//enum of states
{attribute 'strict'}
{attribute 'to_string'}
{attribute 'qualified_only'}
TYPE eTMP :
(
	TotalReset,
	InitCyl,
	InitSrv,
	InitCamQuickFocus,
	InitCamLoadJob,
	Rest,
	SrvPosStart,
	SrvPosStartInterl,
	SrvPosEnd,
	SrvPosEndIntrl,
	CylOut,
	CylIn,
	MtrStartFwd,
	MtrStop,
	MtrStartRev,
	CamReady,
	CamTrig,
	MultiStepTest2,
	MultiStepTest3,
	
	//Example how to use the organiser semi-automode
	//this is a special case in which the operator can choose with a button for example to let the machine do special things 
	//like put servos+clinders automated in a position for configuring/measuring
	
	SemiAutoStart,
	SemiAutoStop
);
END_TYPE

//info on attributes:
//strict 			: don't allow mixing of types
//to_string			: allows the enum to be converted to string
//qualified_only 	: forces the user to start witht the type name (to avoid the situation that accidentially another enum is used)

(* stored: Version 1.1.0.1
   DUT eTMP: Id {943a76cc-00f3-4a33-846d-6a221247c14a} *)
